{attribute 'qualified_only'}
{attribute 'strict'}
TYPE PackMLCommand :
(
	Aborted := 1,
	Clear:= 2, 
	Reset := 3,
	Start := 4
);
END_TYPE

(* stored: Version 1.1.0.1, ProductVersion 3.1.4024.11
   DUT PackMLCommand: Id {487efd2e-ea53-470e-9215-66b5067a1ac5} *)
